Staubli VAL3: CartesianAccel.dtx

public num ca[6]
public num resAccel
